// TIA Portal V20 export
VAR_GLOBAL   // PLC tag table "Default tag table"
   Web_Integer AT %MW10 : Int;
END_VAR
